(* CODESYS project FU_sMidBI.xml

Project tree, tasks and I/O mapping:
  function FU_sMidBI [ST]
*)

// FU_sMidBI
//This functions extracts a part of a string
// |**Version**|**Author**| **Date** |**Changes**
// | 1         | NSN      | 13-06-18 | Creation                                                                                                              |
// | 1.1       | NSN      | 05-02-19 | Made dependant on big output version                                                                                  |
FUNCTION FU_sMidBI : STRING(255)
VAR_IN_OUT
	sStr		:STRING(1);			//Input String
END_VAR
VAR_INPUT
	wLen		:WORD;				//Amount to copy
	wPos		:WORD;				//Position to copy from
END_VAR

FU_sMidBIBO(sOut:= FU_sMidBI,sStr:= sStr,wLen:= wLen,wPos:= wPos,wOutSize:= 255);

END_FUNCTION
